PROGRAM P_VelocityModeTest
VAR
	fbVelocityMode					: VelocityMode;
	fbGetStatusword					: FB_EcCoeSdoRead;
	fbGetActualVelocity				: FB_EcCoeSdoRead;
	bGetStatusword					: BOOL; 
	nTargetVelocity					: DINT;
	nActualVelocity					: DINT;
	nStatusword						: UINT;
	
	bGetActualVelocity				: BOOL;
	fActualVelocityRead				: F_TRIG;
	fStatusWordRead					: F_TRIG;
END_VAR

VAR
	bSetVelocity					: BOOL; 
	bStopMotor						: BOOL;
END_VAR

nTargetVelocity := 200; //rpm
// read FBs
bGetActualVelocity := TRUE;
bGetStatusword := TRUE;


fbGetStatusword(sNetId := GVL.sNetId,
				nSlaveAddr := GVL.nSlaveAddr,
				nIndex := 16#6041,
				nSubindex := 0,
				pDstBuf := ADR(nStatusWord),
				cbBufLen := SIZEOF(nStatusWord),
				bExecute := bGetStatusword);
				
fbGetActualVelocity(sNetId := GVL.sNetId,
					nSlaveAddr := GVL.nSlaveAddr,
					nIndex := 16#6044,
					nSubindex := 0,
					pDstBuf := ADR(nActualVelocity),
					cbBufLen := SIZEOF(nActualVelocity),
					bExecute := bGetActualVelocity);

//set velocity
MAIN.Controlword.4 := 1; //velocity demand value shall equal to ramp output value
MAIN.Controlword.5 := 1; //ramp output value shall follow ramp input value
MAIN.Controlword.6 := 1; //ramp input value shall accord with ramp reference

fbVelocityMode(sNetID := GVL.sNetId,
				nSlaveAddr := GVL.nSlaveAddr,
				nTargetVelocity := nTargetVelocity,
				bSetVelocity := bSetVelocity);
				
//stop
IF bStopMotor THEN
	MAIN.Controlword.8 := 1; //Motor shall be stopped
END_IF
// TODO implement request object 605D<2 velocity deceleration and 605D>=2 quick stop



//reset FBs
fActualVelocityRead.CLK := fbGetActualVelocity.bBusy;
IF fActualVelocityRead.Q THEN
	bGetActualVelocity := FALSE;
END_IF
fStatusWordRead.CLK := fbGetStatusword.bBusy;
IF fStatusWordRead.Q THEN
	bGetStatusword := FALSE;
END_IF

END_PROGRAM

(* stored: Version 1.1.0.1, ProductVersion 3.1.4024.11
   POU P_VelocityModeTest: Id {20dbc57a-bcdc-4d5e-be58-5c2d209d0155}, SpecialFunc None *)
